(* CODESYS project Seminarski.project
   Title: Seminarski
   Version: 0.0.0.0
   Author: Lenovo

Project tree, tasks and I/O mapping:
  MyController : TM241CE24T/U, Schneider Electric, order no. TM241CE24T/U, version 4.0.6.18
    application Application
      libraries: SysTimeRtc, 3.5.1.0 (System)
      task MAST (cyclic, interval 20 ms, priority 15, watchdog 100 ms x 1) calls POU
      global variables GVL
      program POU [ST]
      Symbols
    DI : Digital Inputs, Schneider Electric, version 4.0.6.18
        input  iwDI_IW0 : WORD  // IW0
        input  ibDI_IB1 : BYTE  // IB1
    DQ : Digital Outputs, Schneider Electric, version 4.0.6.18
        output qwDQ_QW0 : WORD  // QW0
        output qbDQ_QB1 : BYTE  // QB1
    Counters : Counters, Schneider Electric, version 4.0.6.18
    Pulse_Generators : Pulse Generators, Schneider Electric, version 4.0.6.18
    Cartridge_1 : Cartridge, Schneider Electric, version 4.0.6.18
    IO_Bus : IO bus - TM3, Schneider Electric, version 4.0.6.18
    COM_Bus : COM bus, Schneider Electric, version 4.0.6.18
    Ethernet_1 : Ethernet Network, Schneider Electric, version 4.0.6.18
    Serial_Line_1 : Serial line, Schneider Electric, version 4.0.6.18
      SoMachine_Network_Manager : SoMachine-Network Manager, Schneider Electric, version 4.0.0.2
    Serial_Line_2 : Serial line, Schneider Electric, version 4.0.6.18
      Modbus_Manager : Modbus Manager, Schneider Electric, version 4.0.0.2
  HMIS5T : HMIS5T, Schneider Electric, order no. HMIS5T, version 3.5.3.54
    HMI Application
    COM1
      SoMachine_Network_Manager1 : SoMachine-Network Manager, Schneider Electric, version 4.0.0.2
    Ethernet
      SoMachine_Network_Manager2 : SoMachine-Network Manager, Schneider Electric, version 4.0.0.2
    USB
      SoMachine_Network_Manager3 : SoMachine-Network Manager, Schneider Electric, version 4.0.0.2
  Vijeo Designer Project Container Data
  Vijeo Designer Project Container
*)

// MyController/Application/GVL
VAR_GLOBAL
END_VAR
VAR_GLOBAL
	mod_rada: UINT := 0;
	I1: BOOL;
	I2: BOOL;
	I3: BOOL;
	I4: BOOL;
	I5: BOOL;
	I6: BOOL;
	I7: BOOL;
	I8: BOOL;
	I9: BOOL;
	I10: BOOL;
	Q1: BOOL;
	Q2: BOOL;
	Q3: BOOL;
	Q4: BOOL;
	Q5: BOOL;
	Q6: BOOL;
	Q7: BOOL;
	Q8: BOOL;
	Q9: BOOL;
	Q10: BOOL;
	reset1: UINT;
	reset2: UINT;
	a: BOOL;
	sat1: UINT;
	minuta1: UINT;
	sekunda1: UINT;
	sat2: UINT;
	minuta2: UINT;
	sekunda2: UINT;
	trenutno_vrijeme: RTS_SYSTIMEDATE;
	STRG: DWORD;
	flag1: UDINT;
	flag2: UDINT;
	pDate: RTS_SYSTIMEDATE;
	broj_sekundi1: UINT;
	broj_sekundi2: UINT;
	broj_sekundi_trenutno: UINT;
END_VAR

// MyController/Application/POU
PROGRAM POU
VAR
	end: INT;
END_VAR

(* Ocitavanje realnog vremena iz biblioteke SysTimeRtc *)
STRG := SysTimeRtcGet(flag1); (* BROJ SEKUNDI PROTEKLIH OD 1.1.1970. *)
flag2 := SysTimeRtcConvertUtcToDate(STRG,pDate);

(* Postavljanje trenutnog vrmena *)
trenutno_vrijeme.wHour := pDate.wHour + 2;
trenutno_vrijeme.wMinute := pDate.wMinute;
trenutno_vrijeme.wSecond := pDate.wSecond;

broj_sekundi1 := (sat1*60*60) + (minuta1*60) + sekunda1;
broj_sekundi2 := (sat2*60*60) + (minuta2*60) + sekunda2;
broj_sekundi_trenutno := (trenutno_vrijeme.wHour*60*60) + (trenutno_vrijeme.wMinute*60) + trenutno_vrijeme.wSecond;

(* Manuelni mod rada *)
IF(mod_rada = 1) THEN
	Q1 := I1;
	Q2 := I2;
	Q3 := I3;
	Q4 := I4;
	Q5 := I5;
	Q6 := I6;
	Q7 := I7;
	Q8 := I8;
	Q9 := I9;
	Q10 := I10;
END_IF 

(* Automatski mod rada *)
IF(mod_rada = 2) THEN
	IF((broj_sekundi_trenutno >= broj_sekundi1) AND (broj_sekundi_trenutno <= broj_sekundi2)) THEN
		Q1 := TRUE;
		Q2 := TRUE;
		Q3 := TRUE;
		Q4 := TRUE;
		Q5 := TRUE;
		Q6 := TRUE;
		Q7 := TRUE;
		Q8 := TRUE;
		Q9 := TRUE;
		Q10 := TRUE;
	ELSE
		Q1 := FALSE;
		Q2 := FALSE;
		Q3 := FALSE;
		Q4 := FALSE;
		Q5 := FALSE;
		Q6 := FALSE;
		Q7 := FALSE;
		Q8 := FALSE;
		Q9 := FALSE;
		Q10 := FALSE;
	END_IF
END_IF

(* Reset koji se desava izmedju manuelnog i automatskog moda *)
IF(a = TRUE AND (reset1 = 1 OR reset2 = 1)) THEN
	Q1 := FALSE;
	Q2 := FALSE;
	Q3 := FALSE;
	Q4 := FALSE;
	Q5 := FALSE;
	Q6 := FALSE;
	Q7 := FALSE;
	Q8 := FALSE;
	Q9 := FALSE;
	Q10 := FALSE;
END_IF

END_PROGRAM
